// TIA Portal V19 export
FUNCTION_BLOCK "F_Zone23_FB"   // FB171, F_LAD
TITLE = SAFETY ZONE 23 - AREA 03 (BORDATRICE)
// -
// stored: Access Published
   VAR
      FNS : "ForceNormalStop";
      F_Contactor_CambioFormato_Bordatrice { ExternalAccessible := 'False'; ExternalVisible := 'False'; ExternalWritable := 'False'} : "FDevice_Contactor_FB";
      F_Sinamics_Bordatrice : "FDevice_Sinamics_FB";
      F_Sinamics_BordatriceCassetta : "FDevice_Sinamics_FB";
   END_VAR
   VAR_TEMP
      DoorNormalStop : Bool;
      DoorSafeStop : Bool;
      Door_Ok : Bool;
   END_VAR
BEGIN

REGION Network 1: < < < < < < < < < < DOOR > > > > > > > > > >
END_REGION

REGION Network 2: Zone Entry enable
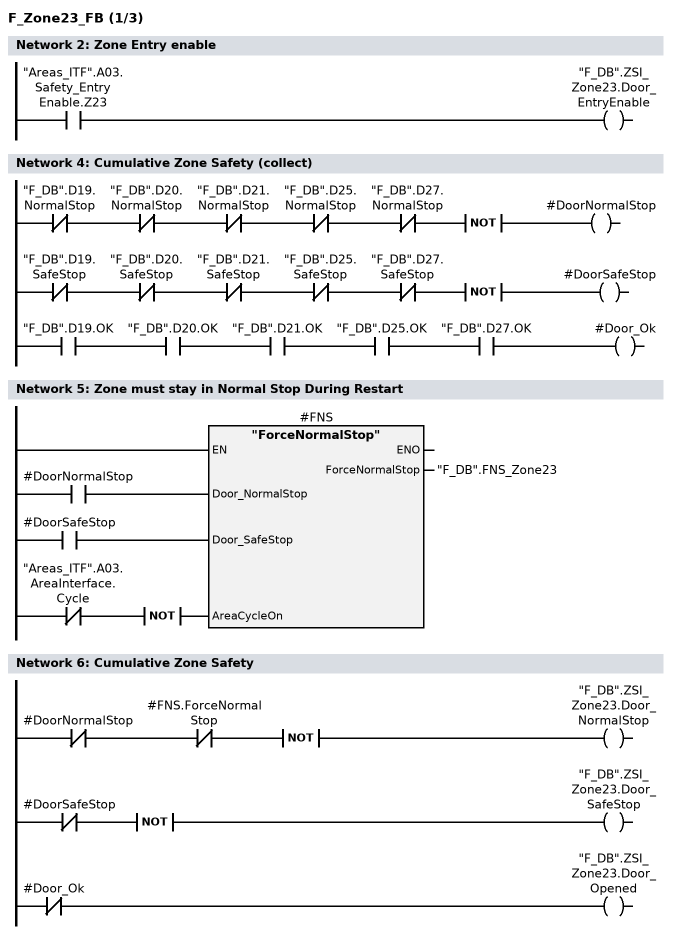
   RUNG wire#powerrail
      Contact( "Areas_ITF".A03.Safety_EntryEnable.Z23 )
      Coil( "F_DB".ZSI_Zone23.Door_EntryEnable )
   END_RUNG
   // the same network as SCL:
   "F_DB".ZSI_Zone23.Door_EntryEnable := "Areas_ITF".A03.Safety_EntryEnable.Z23;
END_REGION

REGION Network 3: < < < < < < < < < < ZONE SAFETY INTERFACE > > > > > > > > > >
END_REGION

REGION Network 4: Cumulative Zone Safety (collect)
   RUNG wire#powerrail
      I_Contact( "F_DB".D19.NormalStop )
      I_Contact( "F_DB".D20.NormalStop )
      I_Contact( "F_DB".D21.NormalStop )
      I_Contact( "F_DB".D25.NormalStop )
      I_Contact( "F_DB".D27.NormalStop )
      Not()
      Coil( #DoorNormalStop )
   END_RUNG
   RUNG wire#powerrail
      I_Contact( "F_DB".D19.SafeStop )
      I_Contact( "F_DB".D20.SafeStop )
      I_Contact( "F_DB".D21.SafeStop )
      I_Contact( "F_DB".D25.SafeStop )
      I_Contact( "F_DB".D27.SafeStop )
      Not()
      Coil( #DoorSafeStop )
   END_RUNG
   RUNG wire#powerrail
      Contact( "F_DB".D19.OK )
      Contact( "F_DB".D20.OK )
      Contact( "F_DB".D21.OK )
      Contact( "F_DB".D25.OK )
      Contact( "F_DB".D27.OK )
      Coil( #Door_Ok )
   END_RUNG
   // the same network as SCL:
   #DoorNormalStop := NOT (NOT "F_DB".D19.NormalStop AND NOT "F_DB".D20.NormalStop AND NOT "F_DB".D21.NormalStop AND NOT "F_DB".D25.NormalStop AND NOT "F_DB".D27.NormalStop);
   #DoorSafeStop := NOT (NOT "F_DB".D19.SafeStop AND NOT "F_DB".D20.SafeStop AND NOT "F_DB".D21.SafeStop AND NOT "F_DB".D25.SafeStop AND NOT "F_DB".D27.SafeStop);
   #Door_Ok := "F_DB".D19.OK AND "F_DB".D20.OK AND "F_DB".D21.OK AND "F_DB".D25.OK AND "F_DB".D27.OK;
END_REGION

REGION Network 5: Zone must stay in Normal Stop During Restart
   RUNG wire#powerrail
      #FNS(Door_NormalStop := wire#w1, Door_SafeStop := wire#w2, AreaCycleOn := wire#w3, ForceNormalStop => "F_DB".FNS_Zone23)
   END_RUNG
   RUNG wire#powerrail
      Contact( #DoorNormalStop )
   END_RUNG wire#w1
   RUNG wire#powerrail
      Contact( #DoorSafeStop )
   END_RUNG wire#w2
   RUNG wire#powerrail
      I_Contact( "Areas_ITF".A03.AreaInterface.Cycle )
      Not()
   END_RUNG wire#w3
   // the same network as SCL:
   #FNS(Door_NormalStop := #DoorNormalStop,   // "ForceNormalStop"
        Door_SafeStop := #DoorSafeStop,
        AreaCycleOn := NOT (NOT "Areas_ITF".A03.AreaInterface.Cycle),
        ForceNormalStop => "F_DB".FNS_Zone23);
END_REGION

REGION Network 6: Cumulative Zone Safety
   RUNG wire#powerrail
      I_Contact( #DoorNormalStop )
      I_Contact( #FNS.ForceNormalStop )
      Not()
      Coil( "F_DB".ZSI_Zone23.Door_NormalStop )
   END_RUNG
   RUNG wire#powerrail
      I_Contact( #DoorSafeStop )
      Not()
      Coil( "F_DB".ZSI_Zone23.Door_SafeStop )
   END_RUNG
   RUNG wire#powerrail
      I_Contact( #Door_Ok )
      Coil( "F_DB".ZSI_Zone23.Door_Opened )
   END_RUNG
   // the same network as SCL:
   "F_DB".ZSI_Zone23.Door_NormalStop := NOT (NOT #DoorNormalStop AND NOT #FNS.ForceNormalStop);
   "F_DB".ZSI_Zone23.Door_SafeStop := NOT (NOT #DoorSafeStop);
   "F_DB".ZSI_Zone23.Door_Opened := NOT #Door_Ok;
END_REGION

REGION Network 7: >
END_REGION

REGION Network 8: >
END_REGION

REGION Network 9: < < < < < < < < < < DEVICES SAFETY VALVES > > > > > > > > > >
END_REGION

REGION Network 10: >
END_REGION

REGION Network 11: >
END_REGION

REGION Network 12: < < < < < < < < < < DEVICES CONTACTORS > > > > > > > > > >
END_REGION

REGION Network 13: Contattore - Cambio formato Bordatrice
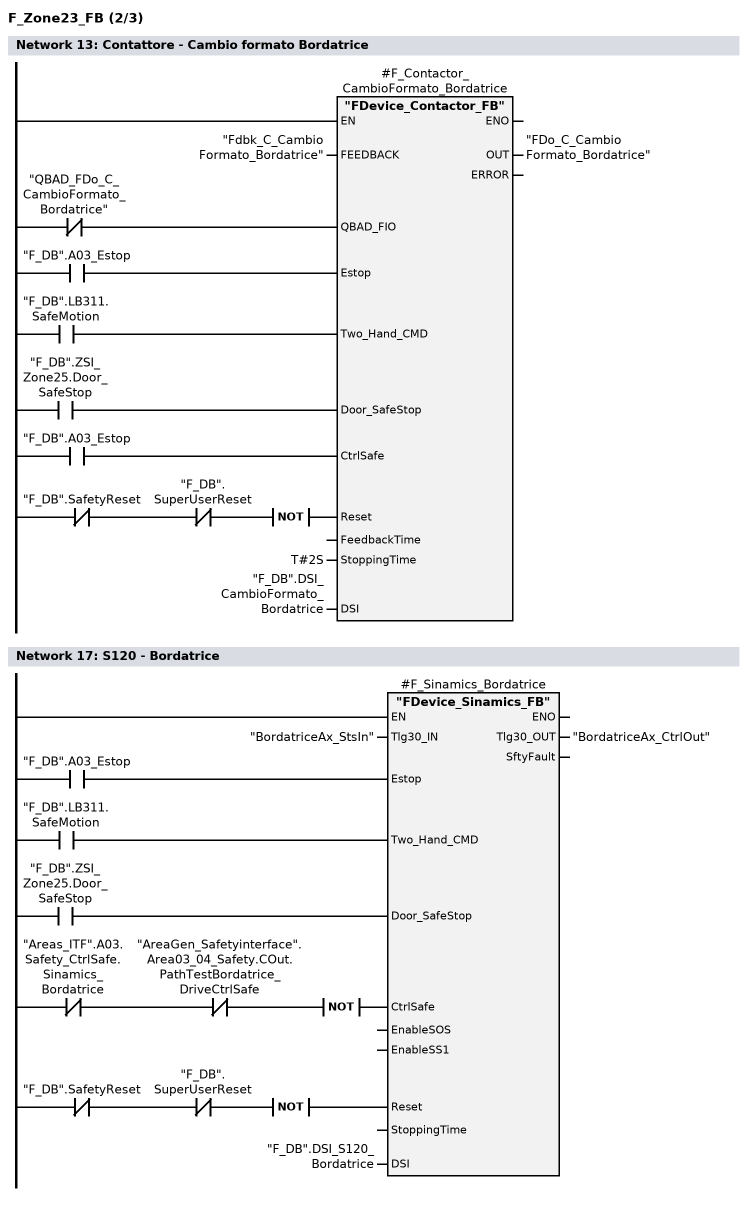
   RUNG wire#powerrail
      #F_Contactor_CambioFormato_Bordatrice(QBAD_FIO := wire#w1, Estop := wire#w2, Two_Hand_CMD := wire#w3, Door_SafeStop := wire#w4, CtrlSafe := wire#w5, Reset := wire#w6, FEEDBACK := "Fdbk_C_CambioFormato_Bordatrice", FeedbackTime :=, StoppingTime := T#2S, DSI := "F_DB".DSI_CambioFormato_Bordatrice, OUT => "FDo_C_CambioFormato_Bordatrice", ERROR =>)
   END_RUNG
   RUNG wire#powerrail
      I_Contact( "QBAD_FDo_C_CambioFormato_Bordatrice" )
   END_RUNG wire#w1
   RUNG wire#powerrail
      Contact( "F_DB".A03_Estop )
   END_RUNG wire#w2
   RUNG wire#powerrail
      Contact( "F_DB".LB311.SafeMotion )
   END_RUNG wire#w3
   RUNG wire#powerrail
      Contact( "F_DB".ZSI_Zone25.Door_SafeStop )
   END_RUNG wire#w4
   RUNG wire#powerrail
      Contact( "F_DB".A03_Estop )
   END_RUNG wire#w5
   RUNG wire#powerrail
      I_Contact( "F_DB".SafetyReset )
      I_Contact( "F_DB".SuperUserReset )
      Not()
   END_RUNG wire#w6
   // the same network as SCL:
   #F_Contactor_CambioFormato_Bordatrice(FEEDBACK := "Fdbk_C_CambioFormato_Bordatrice",   // "FDevice_Contactor_FB"
                           QBAD_FIO := NOT "QBAD_FDo_C_CambioFormato_Bordatrice",
                           Estop := "F_DB".A03_Estop,
                           Two_Hand_CMD := "F_DB".LB311.SafeMotion,
                           Door_SafeStop := "F_DB".ZSI_Zone25.Door_SafeStop,
                           CtrlSafe := "F_DB".A03_Estop,
                           Reset := NOT (NOT "F_DB".SafetyReset AND NOT "F_DB".SuperUserReset),
                           StoppingTime := T#2S,
                           DSI := "F_DB".DSI_CambioFormato_Bordatrice,
                           OUT => "FDo_C_CambioFormato_Bordatrice");
END_REGION

REGION Network 14: >
END_REGION

REGION Network 15: >
END_REGION

REGION Network 16: < < < < < < < < < < DEVICES S120 > > > > > > > > > >
END_REGION

REGION Network 17: S120 - Bordatrice
   RUNG wire#powerrail
      #F_Sinamics_Bordatrice(Estop := wire#w1, Two_Hand_CMD := wire#w2, Door_SafeStop := wire#w3, CtrlSafe := wire#w4, Reset := wire#w5, Tlg30_IN := "BordatriceAx_StsIn", EnableSOS :=, EnableSS1 :=, StoppingTime :=, DSI := "F_DB".DSI_S120_Bordatrice, Tlg30_OUT => "BordatriceAx_CtrlOut", SftyFault =>)
   END_RUNG
   RUNG wire#powerrail
      Contact( "F_DB".A03_Estop )
   END_RUNG wire#w1
   RUNG wire#powerrail
      Contact( "F_DB".LB311.SafeMotion )
   END_RUNG wire#w2
   RUNG wire#powerrail
      Contact( "F_DB".ZSI_Zone25.Door_SafeStop )
   END_RUNG wire#w3
   RUNG wire#powerrail
      I_Contact( "Areas_ITF".A03.Safety_CtrlSafe.Sinamics_Bordatrice )
      I_Contact( "AreaGen_Safetyinterface".Area03_04_Safety.COut.PathTestBordatrice_DriveCtrlSafe )
      Not()
   END_RUNG wire#w4
   RUNG wire#powerrail
      I_Contact( "F_DB".SafetyReset )
      I_Contact( "F_DB".SuperUserReset )
      Not()
   END_RUNG wire#w5
   // the same network as SCL:
   #F_Sinamics_Bordatrice(Tlg30_IN := "BordatriceAx_StsIn",   // "FDevice_Sinamics_FB"
                          Estop := "F_DB".A03_Estop,
                          Two_Hand_CMD := "F_DB".LB311.SafeMotion,
                          Door_SafeStop := "F_DB".ZSI_Zone25.Door_SafeStop,
                          CtrlSafe := NOT (NOT "Areas_ITF".A03.Safety_CtrlSafe.Sinamics_Bordatrice AND NOT "AreaGen_Safetyinterface".Area03_04_Safety.COut.PathTestBordatrice_DriveCtrlSafe),
                          Reset := NOT (NOT "F_DB".SafetyReset AND NOT "F_DB".SuperUserReset),
                          DSI := "F_DB".DSI_S120_Bordatrice,
                          Tlg30_OUT => "BordatriceAx_CtrlOut");
END_REGION

REGION Network 18: S120 - BordatriceCassetta
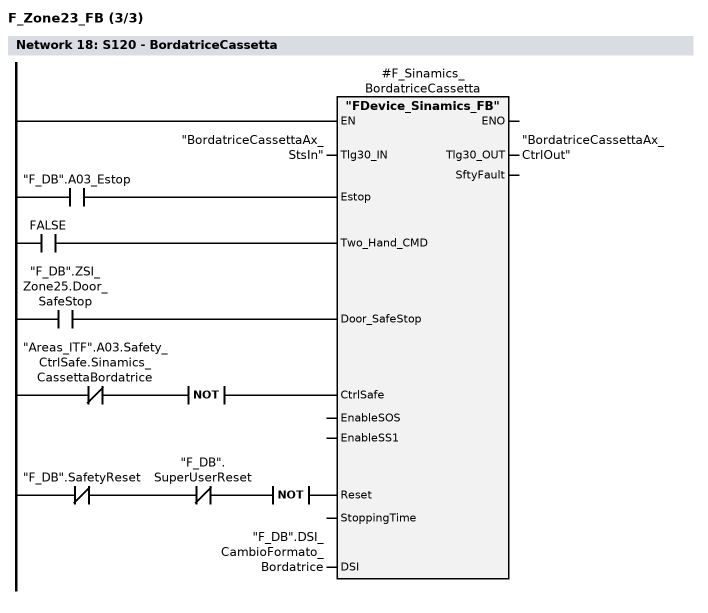
   RUNG wire#powerrail
      #F_Sinamics_BordatriceCassetta(Estop := wire#w1, Two_Hand_CMD := wire#w2, Door_SafeStop := wire#w3, CtrlSafe := wire#w4, Reset := wire#w5, Tlg30_IN := "BordatriceCassettaAx_StsIn", EnableSOS :=, EnableSS1 :=, StoppingTime :=, DSI := "F_DB".DSI_CambioFormato_Bordatrice, Tlg30_OUT => "BordatriceCassettaAx_CtrlOut", SftyFault =>)
   END_RUNG
   RUNG wire#powerrail
      Contact( "F_DB".A03_Estop )
   END_RUNG wire#w1
   RUNG wire#powerrail
      Contact( FALSE )
   END_RUNG wire#w2
   RUNG wire#powerrail
      Contact( "F_DB".ZSI_Zone25.Door_SafeStop )
   END_RUNG wire#w3
   RUNG wire#powerrail
      I_Contact( "Areas_ITF".A03.Safety_CtrlSafe.Sinamics_CassettaBordatrice )
      Not()
   END_RUNG wire#w4
   RUNG wire#powerrail
      I_Contact( "F_DB".SafetyReset )
      I_Contact( "F_DB".SuperUserReset )
      Not()
   END_RUNG wire#w5
   // the same network as SCL:
   #F_Sinamics_BordatriceCassetta(Tlg30_IN := "BordatriceCassettaAx_StsIn",   // "FDevice_Sinamics_FB"
                           Estop := "F_DB".A03_Estop,
                           Two_Hand_CMD := FALSE,
                           Door_SafeStop := "F_DB".ZSI_Zone25.Door_SafeStop,
                           CtrlSafe := NOT (NOT "Areas_ITF".A03.Safety_CtrlSafe.Sinamics_CassettaBordatrice),
                           Reset := NOT (NOT "F_DB".SafetyReset AND NOT "F_DB".SuperUserReset),
                           DSI := "F_DB".DSI_CambioFormato_Bordatrice,
                           Tlg30_OUT => "BordatriceCassettaAx_CtrlOut");
END_REGION

REGION Network 19: >
END_REGION
END_FUNCTION_BLOCK
